Universal Robots URScript: Fase3.script

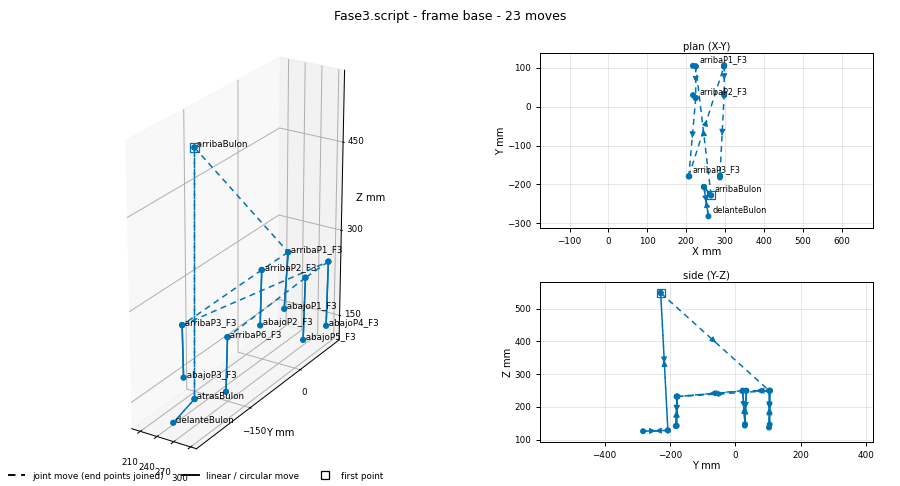
[picture p0: tool path of Fase3.script in frame base, 23 of 24 moves have a stored position in this frame; points joined in program order, loops and branches not executed]
def Fase3():
  set_tool_communication(True, 1000000, 2, 1, 1.5, 3.5)
  set_tool_output_mode(0)
  set_tool_digital_output_mode(0, 1)
  set_tool_digital_output_mode(1, 1)
  set_tool_voltage(0)
  set_safety_mode_transition_hardness(1)
  set_standard_analog_input_domain(0, 1)
  set_standard_analog_input_domain(1, 1)
  set_tool_analog_input_domain(0, 1)
  set_tool_analog_input_domain(1, 1)
  set_analog_outputdomain(0, 0)
  set_analog_outputdomain(1, 0)
  set_input_actions_to_default()
  set_tcp(p[0.00755148296704608,0.003639298738154023,0.026409592411711,0.0,0.0,0.0])
  set_payload(1.14, [0.022, -0.007, 0.054])
  set_gravity([0.0, 0.0, 9.82])
  step_count_833a9f29_8450_4b32_8ecf_da8deb8df3a1 = 0.0
  thread Step_Counter_Thread_0190bdf0_45ae_4d0e_b5b2_50c915833671():
    while (True):
      step_count_833a9f29_8450_4b32_8ecf_da8deb8df3a1 = step_count_833a9f29_8450_4b32_8ecf_da8deb8df3a1 + 1.0
      sync()
    end
  end
  run Step_Counter_Thread_0190bdf0_45ae_4d0e_b5b2_50c915833671()
  global Mesa=p[-0.3283222416297581,-0.20095078680444134,-0.01154506462095492,-2.1087277613487028,-2.3273776320839428,-7.166709239352482E-4]
  # begin: URCap Installation Node
  #   Source: Remote TCP & Toolpath, 1.2.65.build36, Universal Robots A/S
  #   Type: Remote TCP & Toolpath
  # end: URCap Installation Node
  # begin: URCap Installation Node
  #   Source: OnRobot, 5.1.6, OnRobot A/S
  #   Type: Configuración de OnRobot
  on_robot_type = 3
  on_robot_cycle = 2.0
  on_device_ip = "localhost"
  on_device_socket_port = 51234
  on_xmlrpc = rpc_factory("xmlrpc", "http://localhost:41414")
  on_RPC = rpc_factory("xmlrpc", "http://127.0.0.1:31416")
  ON_DEBUG_LOG = False
  on_isMetric = True
  on_toolConnector = True
  on_ioqc = False
  on_dual = False
  on_ft = False
  on_hex = False
  on_gecko = 0
  on_gripper = [False, False, False]
  #======    OnRobot Globals    ======#

  ON_MATH_PI=3.141593
  ON_ZEROPOSE=p[0.0,0.0,0.0,0.0,0.0,0.0]
  ON_ZEROFRAME=p[0.0,0.0,0.0,0.0,0.0,0.0]
  ON_ZERO3D=[0.0,0.0,0.0]
  ON_ZERO6D=[0.0,0.0,0.0,0.0,0.0,0.0]
  ON_ZERO8D=[0.0,0.0,0.0,0.0,0.0,0.0,0.0,0.0]
  ON_FALSE3D=[False,False,False]
  ON_FALSE6D=[False,False,False,False,False,False]
  ON_FALSE8D=[False,False,False,False,False,False,False,False]
  global on_return=0
  on_speedL=ON_ZERO6D
  on_speedBase=ON_ZERO6D
  on_speedVect=ON_ZERO6D
  on_speedExtra=ON_ZERO6D
  on_speedDC=ON_ZERO6D
  on_speedGecko=ON_ZERO6D
  on_floatRegShift=24
  on_intRegShift=24
  on_boolRegShift=64
  ON_BASE_SHIFT_FLOAT=24
  ON_BASE_SHIFT_INT=24
  ON_BASE_SHIFT_BOOL=64
  ON_DEVICE_SHIFT_FLOAT=3
  ON_DEVICE_SHIFT_INT=2
  ON_DEVICE_SHIFT_BOOL=7
  ON_COMMON_SHIFT_FLOAT=12
  ON_COMMON_SHIFT_INT=3
  ON_COMMON_SHIFT_BOOL=1
  ON_DI_SINGLE=0
  ON_DI_PRIMARY=1
  ON_DI_SECONDARY=2
  ON_DI_DUAL=3
  ON_DEVICE_ID_MISSING=0
  ON_INIT_TIMEOUT=500
  on_robot_TCP_offset=ON_ZEROFRAME
  on_tcp_offset_actual=ON_ZEROFRAME
  on_cog_actual=ON_ZEROFRAME
  on_mass_actual=0.0
  on_robot_mount=[0.0,0.0]

  #======    End of OnRobot Globals    ======#
  #======    OnRobot Interface Messages    ======#

  on_devices_primary_log="Dispositivos de OnRobot"
  on_devices_secondary_log="Dispositivo secundario de OnRobot"
  on_device_error_title="OnRobot - Error de dispositivo"
  on_install_error="La configuración de OnRobot no es correcta.<br>Compruebe el estado en la página de configuración de OnRobot, en la pestaña de instalación.<br>Programa detenido."
  on_device_missing="No hay ningún dispositivo conectado.<br>Programa detenido."
  ft_device_missing="No hay ningún sensor F/T OnRobot conectado.<br>Programa detenido."
  rg2ft_device_missing="No hay ninguna pinza RG2-FT conectada.<br>Programa detenido."
  rg_device_missing="No hay ninguna pinza RG conectada.<br>Programa detenido."
  vg_device_missing="No hay ninguna pinza VG conectada.<br>Programa detenido."
  gg_device_missing="No hay ninguna Gecko Gripper conectada.<br>Programa detenido."
  sg_device_missing="No hay ninguna Soft Gripper conectada.<br>Programa detenido."
  tfg_device_missing="No hay ninguna pinza 3FG conectada.<br>Programa detenido."
  on_xmlrpc_start_ip="Conexión al servidor XML-RPC de OnRobot:"
  on_java_comm_error_textmsg_title="OnRobot - Error de comunicación:"
  on_java_comm_controlsocket_open_error="Apertura de la toma 'javaSocket' incorrecta."
  on_java_comm_error_title="OnRobot - Error de comunicación"
  on_java_comm_socket_open_error="El establecimiento de la conexión con el URCap ha excedido el tiempo.<br>Compruebe el estado en la página de configuración de OnRobot, en la pestaña de instalación.<br>Programa detenido."
  on_rtde_feed_error_textmsg_title="OnRobot - Error de comunicación:"
  on_rtde_feed_open_error_textmsg="Apertura de la toma 'rtdeFeed' incorrecta."
  on_rtde_feed_error_title="OnRobot - Error de comunicación"
  on_rtde_feed_open_error="El establecimiento de la conexión con los dispositivos ha excedido el tiempo.<br>Asegúrese de que los dispositivos de OnRobot funcionen y compruebe el estado en la página de configuración de OnRobot, en la pestaña de instalación."

  #======    End of OnRobot Interface Messages    ======#
  #======    OnRobot Interface    ======#

  on_portopened_javaSocket=False
  on_rtde_feed_opened=False
  on_dataRead_running=False
  FT_SENSOR_ID_UNDEFINED=0
  FT_SENSOR_ID_UNKNOWN=1
  FT_SENSOR_ID_HEX_V1=11
  FT_SENSOR_ID_HEX_V2=12
  FT_SENSOR_ID_HEX_V3=13
  FT_SENSOR_ID_RG2FT_V0=20
  FT_SENSOR_ID_RG2FT_V1=21
  FT_SENSOR_ID_RG2FT_V2=22
  def on_error(status_flag,message,title,stop_var=False):
  if(status_flag):
  popup(message,title=title,error=True,blocking=False)
  stop_var=True
  end
  return stop_var
  end
  def on_warning(status_flag,message,title):
  if(status_flag):
  textmsg(title,message)
  end
  end
  def on_missing():
  popup(on_device_missing,title=on_device_error_title,error=True,blocking=False)
  halt
  end
  def ft_missing():
  popup(ft_device_missing,title=on_device_error_title,error=True,blocking=False)
  halt
  end
  def rg2ft_missing():
  popup(rg2ft_device_missing,title=on_device_error_title,error=True,blocking=False)
  halt
  end
  def rg_missing():
  popup(rg_device_missing,title=on_device_error_title,error=True,blocking=False)
  halt
  end
  def vg_missing():
  popup(vg_device_missing,title=on_device_error_title,error=True,blocking=False)
  halt
  end
  def gg_missing():
  popup(gg_device_missing,title=on_device_error_title,error=True,blocking=False)
  halt
  end
  def sg_missing():
  popup(sg_device_missing,title=on_device_error_title,error=True,blocking=False)
  halt
  end
  def tfg_missing():
  popup(tfg_device_missing,title=on_device_error_title,error=True,blocking=False)
  halt
  end
  def on_portclose_javaSocket():
  socket_close("javaSocket")
  on_portopened_javaSocket=False
  end
  def on_portopen_javaSocket():
  on_portclose_javaSocket()
  on_portopened_javaSocket=socket_open("127.0.0.1",44005,"javaSocket")
  if not on_portopened_javaSocket:
  textmsg(on_java_comm_error_textmsg_title,on_java_comm_controlsocket_open_error)
  popup(on_java_comm_socket_open_error,title=on_java_comm_error_title,error=True,blocking=False)
  halt
  end
  end
  def on_rtde_feed_close():
  socket_close("rtdeFeed")
  on_rtde_feed_opened=False
  end
  def on_rtde_feed_open():
  on_rtde_feed_close()
  on_rtde_feed_opened=socket_open(on_device_ip,on_device_socket_port,"rtdeFeed")
  if not on_rtde_feed_opened:
  on_rtde_feed_opened=socket_open(on_device_ip,on_device_socket_port,"rtdeFeed")
  end
  if not on_rtde_feed_opened:
  textmsg(on_rtde_feed_error_textmsg_title,on_rtde_feed_open_error_textmsg)
  popup(on_rtde_feed_open_error,title=on_rtde_feed_error_title,error=True,blocking=False)
  halt
  end
  end
  def on_dataRead():
  enter_critical
  floatRegDummy=read_input_float_register(0+on_floatRegShift)
  on_speedVect[0]=floatRegDummy/1000.0
  floatRegDummy=read_input_float_register(1+on_floatRegShift)
  on_speedVect[1]=floatRegDummy/1000.0
  floatRegDummy=read_input_float_register(2+on_floatRegShift)
  on_speedVect[2]=floatRegDummy/1000.0
  floatRegDummy=read_input_float_register(3+on_floatRegShift)
  on_speedVect[3]=floatRegDummy
  floatRegDummy=read_input_float_register(4+on_floatRegShift)
  on_speedVect[4]=floatRegDummy
  floatRegDummy=read_input_float_register(5+on_floatRegShift)
  on_speedVect[5]=floatRegDummy
  exit_critical
  end
  def on_set_rtde_watchdog(updateHz=5,ftWD=False,gripperWD=-1):
  local update_str=str_cat(" watchdog set to [Hz]: ",updateHz)
  if ftWD:
  watchdog_int_reg_str=str_cat("input_int_register_",0+on_intRegShift)
  rtde_set_watchdog(watchdog_int_reg_str,updateHz,"stop")
  if ON_DEBUG_LOG:
  textmsg(watchdog_int_reg_str,update_str)
  end
  end
  if not(gripperWD<0):
  if(gripperWD==ON_DI_SINGLE or gripperWD==ON_DI_PRIMARY or gripperWD==ON_DI_DUAL):
  watchdog_int_reg_str=str_cat("input_int_register_",3+on_intRegShift)
  rtde_set_watchdog(watchdog_int_reg_str,updateHz,"stop")
  if ON_DEBUG_LOG:
  textmsg(watchdog_int_reg_str,update_str)
  end
  end
  if(gripperWD==ON_DI_SECONDARY or gripperWD==ON_DI_DUAL):
  watchdog_int_reg_str=str_cat("input_int_register_",ON_DEVICE_SHIFT_INT+3+on_intRegShift)
  rtde_set_watchdog(watchdog_int_reg_str,updateHz,"stop")
  if ON_DEBUG_LOG:
  textmsg(watchdog_int_reg_str,update_str)
  end
  end
  end
  end
  def on_speedVect_get():
  return[on_speedVect[0],on_speedVect[1],on_speedVect[2],on_speedVect[3],on_speedVect[4],on_speedVect[5]]
  end
  def on_speedDC_get():
  local speedExtra=ON_ZERO6D
  if on_speedl_for_depthcompensation:
  speedExtra=[on_speedDC[0],on_speedDC[1],on_speedDC[2],on_speedDC[3],on_speedDC[4],on_speedDC[5]]
  end
  return speedExtra
  end
  def on_speedDC_set(speedDC):
  on_speedDC=[speedDC[0],speedDC[1],speedDC[2],speedDC[3],speedDC[4],speedDC[5]]
  end
  def on_speedGecko_get():
  local speedExtra=ON_ZERO6D
  if on_speedl_for_gecko:
  speedExtra=[on_speedGecko[0],on_speedGecko[1],on_speedGecko[2],on_speedGecko[3],on_speedGecko[4],on_speedGecko[5]]
  end
  return speedExtra
  end
  def on_speedGecko_set(speedGecko):
  on_speedGecko=[speedGecko[0],speedGecko[1],speedGecko[2],speedGecko[3],speedGecko[4],speedGecko[5]]
  end
  thread on_dataRead_thread():
  if ON_DEBUG_LOG:
  textmsg("Starting on_dataRead thread")
  end
  while on_dataRead_running:
  sync()
  on_dataRead()
  end
  if ON_DEBUG_LOG:
  textmsg("Stopping on_dataRead thread")
  end
  end

  #======    End of OnRobot Interface    ======#
  #======    OnRobot QC Setup Tool Connector    ======#

  def tc_setup_tool():
  if ON_DEBUG_LOG:
  textmsg("QC Setup Tool Connector start...")
  end
  set_tool_voltage(24)

  set_tool_communication(True,1000000,2,1,1.5,3.5)

  if ON_DEBUG_LOG:
  textmsg("QC Setup Tool Connector end.")
  end
  end

  #======    End of OnRobot QC Setup Tool Connector    ======#
  #======    OnRobot TCP Messages    ======#

  on_tcp_log_msg_default="OnRobot: Desplazamiento del TCP del robot establecido en:"
  on_tcp_log_msg_primary="OnRobot: Desplazamiento del TCP del robot establecido en primario:"
  on_tcp_log_msg_secondary="OnRobot: Desplazamiento del TCP del robot establecido en secundario:"

  #======    End of OnRobot TCP Messages    ======#
  #======    OnRobot TCP    ======#

  on_tcp_offset_actual=ON_ZEROFRAME
  on_tcp_offset_primary=ON_ZEROFRAME
  on_tcp_static_primary=ON_ZEROFRAME
  on_tcp_dynamic_primary=ON_ZEROFRAME
  on_tcp_vision_primary=ON_ZEROFRAME
  on_tcp_qc_primary=ON_ZEROFRAME
  on_tcp_base_primary=ON_ZEROFRAME
  on_tcp_gripper_static_primary=ON_ZEROFRAME
  on_tcp_tool_primary=ON_ZEROFRAME
  on_tcp_gripper_dynamic_primary=ON_ZEROFRAME
  on_tcp_gripper_primary=ON_ZEROFRAME
  on_tcp_offset_secondary=ON_ZEROFRAME
  on_tcp_static_secondary=ON_ZEROFRAME
  on_tcp_dynamic_secondary=ON_ZEROFRAME
  on_tcp_vision_secondary=ON_ZEROFRAME
  on_tcp_qc_secondary=ON_ZEROFRAME
  on_tcp_base_secondary=ON_ZEROFRAME
  on_tcp_gripper_static_secondary=ON_ZEROFRAME
  on_tcp_tool_secondary=ON_ZEROFRAME
  on_tcp_gripper_dynamic_secondary=ON_ZEROFRAME
  on_tcp_gripper_secondary=ON_ZEROFRAME
  def on_tcp_update_primary():
  if ON_DEBUG_LOG:
  textmsg("TCP Update Primary start..")
  end
  on_tcp_gripper_dynamic_primary=p[0.0, 0.0, 0.0, 0.0, 0.0, 0.0]
  enter_critical
  on_tcp_dynamic_primary=pose_trans(on_tcp_static_primary,on_tcp_gripper_dynamic_primary)
  on_tcp_offset_primary=pose_trans(on_tcp_dynamic_primary,on_tcp_tool_primary)
  exit_critical
  if ON_DEBUG_LOG:
  textmsg("TCP Update Primary end.")
  end
  end
  def on_tcp_init_primary():
  if ON_DEBUG_LOG:
  textmsg("TCP Init Primary start..")
  end
  enter_critical
  on_tcp_base_primary=pose_trans(on_tcp_vision_primary,on_tcp_qc_primary)
  on_tcp_static_primary=pose_trans(on_tcp_base_primary,on_tcp_gripper_static_primary)
  exit_critical
  on_tcp_update_primary()
  if ON_DEBUG_LOG:
  textmsg("TCP Init Primary end.")
  end
  end
  def on_tcp_offset_set(TCP_offset):
  if ON_DEBUG_LOG:
  textmsg("TCP Offset set started!")
  end
  on_tcp_offset_send(TCP_offset)
  if(on_follow_tcp):
  set_tcp(TCP_offset)
  end
  on_robot_TCP_offset=TCP_offset
  if ON_DEBUG_LOG:
  textmsg("TCP Offset set to: ",on_robot_TCP_offset)
  end
  end
  def on_tcp_offset_forced_set_actual(isPrimary=True):
  if(not on_follow_tcp):

  local tcp_log_msg=on_tcp_log_msg_default

  textmsg(tcp_log_msg,on_tcp_offset_actual)
  set_tcp(on_tcp_offset_actual)
  end
  end
  def on_tcp_update(isPrimary=True):
  on_tcp_update_primary()

  on_tcp_set_actual_to(isPrimary)
  end
  def on_tcp_set_actual_to(isPrimary=True):

  on_tcp_offset_actual=on_tcp_offset_primary
  if(on_follow_tcp):
  textmsg(on_tcp_log_msg_default,on_tcp_offset_actual)
  end

  on_tcp_active_is_primary=isPrimary
  on_tcp_offset_set(on_tcp_offset_actual)
  end
  def on_tcp_update_tool_primary(tool_offset):
  if ON_DEBUG_LOG:
  textmsg("TCP Update Tool Primary start..")
  end
  on_tcp_tool_primary=tool_offset
  on_tcp_update_primary()
  if ON_DEBUG_LOG:
  textmsg("TCP Update Tool Primary end.")
  end
  end
  def on_tcp_tool_rpy_get(xyz=[0.0,0.0,0.0],rpy=[0.0,0.0,0.0]):
  local rotvec=rpy2rotvec(rpy)
  local tool_offset=p[xyz[0],xyz[1],xyz[2],rotvec[0],rotvec[1],rotvec[2]]
  return tool_offset
  end

  def on_tcp_update_tool(tool_offset,tool_index=0):
  if ON_DEBUG_LOG:
  textmsg("TCP Update Tool start..")
  end
  if(tool_index!=ON_DI_SECONDARY):
  on_tcp_update_tool_primary(tool_offset)
  local isPrimary=True

  end
  on_tcp_set_actual_to(isPrimary)
  if ON_DEBUG_LOG:
  textmsg("TCP Update Tool end.")
  end
  end

  #======    End of OnRobot TCP    ======#
  #======    OnRobot Payload Messages    ======#

  on_mass_log_msg="OnRobot: Masa de la carga útil del robot establecida en:"
  on_cog_log_msg="OnRobot: Centro de gravedad de la carga útil del robot establecido en:"

  #======    End of OnRobot Payload Messages    ======#
  #======    OnRobot Payload    ======#

  on_cog_actual=ON_ZEROFRAME
  on_mass_actual=0.0
  on_cog_primary=ON_ZEROFRAME
  on_cog_L1L2_primary=ON_ZEROFRAME
  on_mass_primary=0.0
  on_mass_L1L2_primary=0.0
  on_cog_vision_primary=ON_ZEROFRAME
  on_cog_qc_primary=ON_ZEROFRAME
  on_cog_base_primary=ON_ZEROFRAME
  on_cog_gripper_primary=ON_ZEROFRAME
  on_cog_tool_primary=ON_ZEROFRAME
  on_mass_vision_primary=0.0
  on_mass_qc_primary=0.0
  on_mass_base_primary=0.0
  on_mass_gripper_primary=0.0
  on_mass_tool_primary=0.0
  on_cog_secondary=ON_ZEROFRAME
  on_mass_secondary=0.0
  on_cog_gripper_secondary=ON_ZEROFRAME
  on_mass_gripper_secondary=0.0
  on_cog_tool_secondary=ON_ZEROFRAME
  on_mass_tool_secondary=0.0
  ON_LB2KG001=0.45359237/100
  def on_payload_update_primary():
  if ON_DEBUG_LOG:
  textmsg("Payload Update Primary start..")
  end
  enter_critical
  on_mass_primary=on_mass_L1L2_primary+on_mass_tool_primary
  local massL1L2L3Ratio=on_mass_tool_primary/on_mass_primary
  local toolAbsCOG=pose_trans(on_tcp_dynamic_primary,on_cog_tool_primary)
  toolAbsCOG=p[toolAbsCOG[0],toolAbsCOG[1],toolAbsCOG[2],0.0,0.0,0.0]
  on_cog_primary=interpolate_pose(on_cog_L1L2_primary,toolAbsCOG,massL1L2L3Ratio)
  on_cog_primary=p[on_cog_primary[0],on_cog_primary[1],on_cog_primary[2],0.0,0.0,0.0]
  exit_critical
  if ON_DEBUG_LOG:
  textmsg("Payload Update Primary end.")
  end
  end
  def on_payload_init_primary():
  if ON_DEBUG_LOG:
  textmsg("Payload Init Primary start..")
  end
  enter_critical
  on_mass_base_primary=on_mass_vision_primary+on_mass_qc_primary
  local massL0L1Ratio=on_mass_qc_primary/on_mass_base_primary
  on_mass_L1L2_primary=on_mass_base_primary+on_mass_gripper_primary
  local massL1L2Ratio=on_mass_gripper_primary/on_mass_L1L2_primary
  local qcAbsCOG=pose_trans(on_tcp_vision_primary,on_cog_qc_primary)
  qcAbsCOG=p[qcAbsCOG[0],qcAbsCOG[1],qcAbsCOG[2],0.0,0.0,0.0]
  on_cog_base_primary=interpolate_pose(on_cog_vision_primary,qcAbsCOG,massL0L1Ratio)
  on_cog_base_primary=p[on_cog_base_primary[0],on_cog_base_primary[1],on_cog_base_primary[2],0.0,0.0,0.0]
  local gripperAbsCOG=pose_trans(on_tcp_base_primary,on_cog_gripper_primary)
  gripperAbsCOG=p[gripperAbsCOG[0],gripperAbsCOG[1],gripperAbsCOG[2],0.0,0.0,0.0]
  on_cog_L1L2_primary=interpolate_pose(on_cog_base_primary,gripperAbsCOG,massL1L2Ratio)
  on_cog_L1L2_primary=p[on_cog_L1L2_primary[0],on_cog_L1L2_primary[1],on_cog_L1L2_primary[2],0.0,0.0,0.0]
  exit_critical
  on_payload_update_primary()
  if ON_DEBUG_LOG:
  textmsg("Payload Init Primary end.")
  end
  end
  def on_payload_update():
  on_payload_update_primary()

  on_mass_actual =on_mass_primary
  on_cog_actual=on_cog_primary

  on_payload_set_actual()
  end
  def on_payload_set_actual():

  on_mass_actual =on_mass_primary
  on_cog_actual=on_cog_primary

  local CoG=[on_cog_actual[0],on_cog_actual[1],on_cog_actual[2]]
  on_payload_set(on_mass_actual,CoG)
  end
  def on_payload_update_tool_primary(tool_mass=0,tool_cog=[0.0,0.0,0.0]):
  if ON_DEBUG_LOG:
  textmsg("Payload Update Tool Primary start..")
  end
  on_cog_tool_primary=p[tool_cog[0],tool_cog[1],tool_cog[2],0.0,0.0,0.0]
  on_mass_tool_primary=tool_mass
  on_payload_update_primary()
  if ON_DEBUG_LOG:
  textmsg("Payload Update Tool Primary end.")
  end
  end
  def on_payload_set(mass,CoG):
  if ON_DEBUG_LOG:
  textmsg("Payload set started!")
  end
  local center_of_gravity=[CoG[0],CoG[1],CoG[2]]
  on_payload_send(center_of_gravity,mass)
  if(on_isMetric):
  local roundedMass=floor(mass*100+0.5)/100
  else:
  local roundedMass=floor(mass/ON_LB2KG001+0.5)*ON_LB2KG001
  end
  set_payload(roundedMass,center_of_gravity)
  on_mass_actual=roundedMass
  on_cog_actual=p[CoG[0],CoG[1],CoG[2],0.0,0.0,0.0]
  if ON_DEBUG_LOG:
  textmsg("Payload mass, CoG set to: ",str_cat(str_cat(mass,", "),CoG))
  end
  end

  def on_payload_update_secondary():
  end
  def on_payload_init_secondary():
  end

  def on_payload_update_tool(tool_mass,tool_cog=[0.0,0.0,0.0],tool_index=0):
  if ON_DEBUG_LOG:
  textmsg("Payload Update Tool start..")
  end
  if(tool_index!=ON_DI_SECONDARY):
  on_cog_tool_primary=p[tool_cog[0],tool_cog[1],tool_cog[2],0.0,0.0,0.0]
  on_mass_tool_primary=tool_mass
  else:
  on_cog_tool_secondary=p[tool_cog[0],tool_cog[1],tool_cog[2],0.0,0.0,0.0]
  on_mass_tool_secondary=tool_mass
  end
  on_payload_update()
  if ON_DEBUG_LOG:
  textmsg("Payload Update Tool end.")
  end
  end
  def on_payload_get_cog2tcp_tool(tool_index=0):
  if(tool_index!=ON_DI_SECONDARY):
  local cog_tool=[on_tcp_tool_primary[0],on_tcp_tool_primary[1],on_tcp_tool_primary[2]]
  else:
  local cog_tool=[on_tcp_tool_secondary[0],on_tcp_tool_secondary[1],on_tcp_tool_secondary[2]]
  end
  return cog_tool
  end

  #======    End of OnRobot Payload    ======#
  #======    OnRobot QC TCP    ======#

  onrobotmini=0

  def on_tcp_offset_send(TCP_offset):
  on_robot_TCP_offset=TCP_offset
  end
  def on_payload_send(CoG,mass):
  on_robot_payload_cog=CoG
  on_robot_payload_mass=mass
  end


  #======    End of OnRobot QC TCP    ======#
  #======    OnRobot  Speedl    ======#

  on_speedl_thread_handler=0
  on_speedl_is_enabled=False
  on_speedl_is_running=False
  on_speedl_acc=0.0
  ft_speedl_hg_caranteen_reached=False
  ft_speedl_hg_caranteen_safemode=False
  on_speedl_for_ftcontrol=False
  on_speedl_for_move=False
  on_speedl_for_handguide=False
  on_speedl_for_insertpart=False
  on_speedl_for_depthcompensation=False
  on_speedl_for_center=False
  on_speedl_for_gecko=False
  on_speedl_acc=10000.0
  on_speedl_acc_to_zero=3.0
  ON_SPEEDL_FTCONTROL=1
  ON_SPEEDL_HANDGUIDE=2
  ON_SPEEDL_MOVE=3
  ON_SPEEDL_INSERTPART=4
  ON_SPEEDL_DEPTHCOMP=5
  ON_SPEEDL_CENTER=6
  ON_SPEEDL_GECKO=7
  def on_speedl_add_extra(speedBase,speedExtra):
  speedSum=ON_ZERO6D
  speedBaseP=p[speedBase[0],speedBase[1],speedBase[2],speedBase[3],speedBase[4],speedBase[5]]
  speedExtraP=p[speedExtra[0],speedExtra[1],speedExtra[2],speedExtra[3],speedExtra[4],speedExtra[5]]
  speedSumP=pose_add(speedExtraP,speedBaseP)
  speedSum=[speedSumP[0],speedSumP[1],speedSumP[2],speedSumP[3],speedSumP[4],speedSumP[5]]
  return speedSum
  end

  thread on_speedl_thread():
  if ON_DEBUG_LOG:
  textmsg("Speedl thread started..")
  end
  enter_critical
  on_speedl_is_running=True
  on_speedl_is_enabled=True
  exit_critical
  on_speedL=ON_ZERO6D

  while on_speedl_is_running:
  on_speedBase=on_speedVect_get()
  on_speedL=on_speedBase



  if on_speedl_is_enabled:
  speedl(on_speedL,a=on_speedl_acc,t=0.001)
  else:
  speedl(ON_ZERO6D,a=on_speedl_acc_to_zero,t=0.001)
  end
  end

  on_speedL=ON_ZERO6D
  if ON_DEBUG_LOG:
  textmsg("Speedl thread ended.")
  end
  end
  def on_speedl_integer_get():
  local speedl_integer=binary_list_to_integer([on_speedl_for_ftcontrol,on_speedl_for_handguide,on_speedl_for_move,on_speedl_for_insertpart,on_speedl_for_depthcompensation,on_speedl_for_center,on_speedl_for_gecko])
  return speedl_integer
  end
  def on_speedl_start_for(speedl_id):
  if(speedl_id==ON_SPEEDL_FTCONTROL):
  on_speedl_for_ftcontrol=True
  elif(speedl_id==ON_SPEEDL_HANDGUIDE):
  on_speedl_for_handguide=True
  elif(speedl_id==ON_SPEEDL_MOVE):
  on_speedl_for_move=True
  elif(speedl_id==ON_SPEEDL_INSERTPART):
  on_speedl_for_insertpart=True
  elif(speedl_id==ON_SPEEDL_DEPTHCOMP):
  on_speedl_for_depthcompensation=True
  elif(speedl_id==ON_SPEEDL_CENTER):
  on_speedl_for_center=True
  elif(speedl_id==ON_SPEEDL_GECKO):
  on_speedl_for_gecko=True
  else:
  textmsg("Unknown Start speedl ID received: ",speedl_id)
  end
  local speedl_integer=on_speedl_integer_get()
  if not(speedl_integer==0):
  if not on_speedl_is_running:
  on_speedl_thread_handler=run on_speedl_thread()
  end
  end
  return on_speedl_is_running
  end
  def on_speedl_stop_for(speedl_id,brake=10):
  if(speedl_id==ON_SPEEDL_FTCONTROL):
  on_speedl_for_ftcontrol=False
  elif(speedl_id==ON_SPEEDL_HANDGUIDE):
  on_speedl_for_handguide=False
  elif(speedl_id==ON_SPEEDL_MOVE):
  on_speedl_for_move=False
  elif(speedl_id==ON_SPEEDL_INSERTPART):
  on_speedl_for_insertpart=False
  elif(speedl_id==ON_SPEEDL_DEPTHCOMP):
  on_speedl_for_depthcompensation=False
  on_speedDC_set(ON_ZERO6D)
  elif(speedl_id==ON_SPEEDL_CENTER):
  on_speedl_for_center=False
  elif(speedl_id==ON_SPEEDL_GECKO):
  on_speedl_for_gecko=False
  on_speedGecko_set(ON_ZERO6D)
  else:
  textmsg("Unknown Stop speedl ID received: ",speedl_id)
  end
  local speedl_integer=on_speedl_integer_get()
  if(speedl_integer==0):
  if(on_speedl_is_running):
  kill on_speedl_thread_handler
  enter_critical
  on_speedl_is_running=False
  exit_critical

  end
  if ON_DEBUG_LOG:
  textmsg("Speedl thread stopped")
  end
  stopl(brake)
  end
  return on_speedl_is_running
  end
  def on_speedl_pause():
  on_speedl_is_enabled=False
  return on_speedl_integer_get()
  end
  def on_speedl_resume():
  on_speedl_is_enabled=True
  return on_speedl_integer_get()
  end
  def on_wait_ms(time_ms):
  local sync_time=ceil(norm(time_ms/2.0))
  while(sync_time>0):
  sync_time=sync_time-1
  sync()
  end
  end

  #======    End of OnRobot  Speedl    ======#
  on_install_tcp = False
  on_follow_tcp = False
  textmsg(on_devices_primary_log, ": Quick Changer + Lado de la herramienta de QC + [0.0, 0.0, 0.0, 0.0, 0.0, 0.0]")
  on_tcp_active_is_primary = True
  on_tcp_vision_primary = p[0.0, 0.0, 0.0, 0.0, 0.0, 0.0]
  on_cog_vision_primary = p[0.0, 0.0, 0.0, 0.0, 0.0, 0.0]
  on_mass_vision_primary = 0.0
  on_tcp_qc_primary = p[0.0, 0.0, 0.0136, 0.0, 0.0, 0.0]
  on_cog_qc_primary = p[0.0, 0.0, 0.004, 0.0, 0.0, 0.0]
  on_mass_qc_primary = 0.06
  on_tcp_gripper_static_primary = p[0.0, 0.0, 0.017, 0.0, 0.0, 0.0]
  on_cog_gripper_primary = p[0.0, 0.0, 0.002, 0.0, 0.0, 0.0]
  on_mass_gripper_primary = 0.14
  on_tcp_tool_primary = p[0.0, 0.0, 0.0, 0.0, 0.0, 0.0]
  on_cog_tool_primary = p[0.0, 0.0, 0.0, 0.0, 0.0, 0.0]
  on_mass_tool_primary = 0.0
  #======    OnRobot Run    ======#

  textmsg(on_xmlrpc_start_ip,on_device_ip)
  on_portopen_javaSocket()
  sync()
  on_rtde_feed_open()
  sync()
  local gripperWDs=binary_list_to_integer(on_gripper)
  if gripperWDs==0:
  gripperWDs=-1
  else:
  gripperWDs=floor(gripperWDs/2)
  end
  on_set_rtde_watchdog(updateHz=0.2,ftWD=on_ft,gripperWD=gripperWDs)
  sync()
  on_dataRead_running=True
  sync()
  on_dataRead_thrd=run on_dataRead_thread()
  sync()
  on_tcp_init_primary()
  on_payload_init_primary()

  on_tcp_set_actual_to(on_tcp_active_is_primary)
  if(on_follow_tcp):
  on_payload_set_actual()
  end

  #======    End of OnRobot Run    ======#
  #======    OnRobot QC Start    ======#

  if(on_toolConnector):
  tc_setup_tool()
  end
  sync()

  #======    End of OnRobot QC Start    ======#
  # end: URCap Installation Node
  global arribaBulon_p=p[.264097371719, -.228254341384, .548494258749, 1.585288091520, .085368942758, .052684265010]
  global arribaBulon_q=[0.0823671817779541, -1.5479493898204382, -0.842977762222274, -2.249339719811945, 0.01133561134338383, -1.6629841963397176]
  global atrasBulon_p=p[.245619565393, -.206229029031, .127949595254, 1.145266979799, 1.284974715224, -1.172261599952]
  global atrasBulon_q=[0.18570303241219666, -1.8425440913304127, -2.1757274455361326, -2.137330201992251, 0.1096066770252433, -1.7350318094075643]
  global delanteBulon_p=p[.257367062930, -.282169444566, .125542628574, 1.158631853822, 1.223105278388, -1.250786556870]
  global delanteBulon_q=[-0.127409035395587, -2.02615272864022, -1.95040543910366, -2.0546015954477355, -0.14137166941154078, -1.8664551020827291]
  global arribaP1_F3_p=p[.224644079235, .103836313498, .249354312056, -2.208051583079, -2.214597805453, .012045887033]
  global arribaP1_F3_q=[0.9707521299592239, -1.174781119517391, -2.0064305080926808, -1.5350170771289937, 1.5830136315588959, -2.1699678590045597]
  global abajoP1_F3_p=p[.217351130895, .105158373635, .145871126277, -2.208007269394, -2.214589077087, .011773755537]
  global abajoP1_F3_q=[1.0053096491487898, -1.3109168011728976, -2.4436354857172944, -0.9609782861480696, 1.5838862961847608, -2.1366320702914097]
  global arribaP2_F3_p=p[.224582479854, .022513190074, .249352391909, -2.207989835995, -2.214569210422, .012088793108]
  global arribaP2_F3_q=[0.6852162643329649, -1.0683160351457337, -2.0586158527273106, -1.5934856070708179, 1.5814428352320764, -2.455329191705632]
  global abajoP2_F3_p=p[.217746809497, .029725857966, .147153686199, -2.207987963195, -2.214642841298, .012082484581]
  global abajoP2_F3_q=[0.7419977188110352, -1.1732912820628645, -2.511789321899414, -1.0345638555339338, 1.5826172828674319, -2.399748627339495]
  global arribaP3_F3_p=p[.206750338136, -.179228225553, .231443959029, -2.197588078884, 2.235277736991, -.020786326198]
  global arribaP3_F3_q=[-0.18465583486099035, -1.3281955607676812, -2.0006709215611025, -1.3676400018627604, 1.5652112731884946, -0.1644100155378494]
  global abajoP3_F3_p=p[.208204529507, -.179202485408, .142240823155, -2.197553268895, 2.235243844556, -.020796942752]
  global abajoP3_F3_q=[-0.18301994005315336, -1.5208934110454173, -2.310643196105966, -0.8649354738047563, 1.565710783004826, -0.16392451921577944]
  global arribaP4_F3_p=p[.297933427712, .105957309290, .249359521855, -2.208163486704, -2.214602719616, .012089079617]
  global arribaP4_F3_q=[0.7490953149560091, -1.5138985931798459, -1.7521360360771503, -1.4535102010608423, 1.5802211047555632, -2.392322805708589]
  global abajoP4_F3_p=p[.297416304891, .103134700907, .136772641869, -2.207987172695, -2.214699703310, .011928594507]
  global abajoP4_F3_q=[0.7431611954992511, -1.7071065413756177, -2.13331594471272, -0.8791223442295077, 1.5809192364563067, -2.3998277214921577]
  global arribaP5_F3_p=p[.297927188132, .033813878502, .249377734153, -2.208173548754, -2.214589723707, .011925302641]
  global arribaP5_F3_q=[0.5391322059410543, -1.4463543511276873, -1.8116517635701346, -1.4641567094980132, 1.5784757755036594, -2.6021113817983164]
  global abajoP5_F3_p=p[.297930409515, .029154935950, .142651108607, -2.208220572640, -2.214607723347, .011878116817]
  global abajoP5_F3_q=[0.524354457855229, -1.6304494343199663, -2.1841697692871014, -0.907690839176535, 1.5789034366607568, -2.6182459036456485]
  global arribaP6_F3_p=p[.286922377788, -.177452737853, .231463994865, -2.197503334999, 2.235293632857, -.020976529593]
  global arribaP6_F3_q=[-0.13142329267507336, -1.6315337847643132, -1.7285740911751137, -1.3363986082522743, 1.5632914110110594, -0.11187560505271055]
  global abajoP6_F3_p=p[.286936793143, -.182063295540, .141255559416, -2.197478510061, 2.235221511214, -.020803429330]
  global abajoP6_F3_q=[-0.1460840583919243, -1.8058921770385403, -1.9922933411515018, -0.8983209660015365, 1.564164075637315, -0.12775810124598674]
  $ 1 "Robot Program"
  $ 2 "Set DO[0]=Apagar"
  set_standard_digital_out(0, False)
  $ 3 "i≔1"
  global i=1
  $ 4 "Loop i≤6"
  while (i <= 6):
    $ 5 "MoveJ"
    $ 6 "arribaBulon" "breakAfter"
    movej(get_inverse_kin(arribaBulon_p, qnear=arribaBulon_q), a=1.2, v=0.75)
    $ 7 "MoveJ"
    $ 8 "atrasBulon" "breakAfter"
    movej(get_inverse_kin(atrasBulon_p, qnear=atrasBulon_q), a=1.2, v=0.75)
    $ 9 "MoveJ"
    $ 10 "delanteBulon" "breakAfter"
    movej(get_inverse_kin(delanteBulon_p, qnear=delanteBulon_q), a=1.3962634015954636, v=1.0471975511965976)
    $ 11 "Set DO[0]=Encender"
    set_standard_digital_out(0, True)
    $ 12 "Wait: 0.25"
    sleep(0.25)
    $ 13 "MoveJ"
    $ 14 "atrasBulon" "breakAfter"
    movej(get_inverse_kin(atrasBulon_p, qnear=atrasBulon_q), a=1.3962634015954636, v=1.0471975511965976)
    $ 15 "MoveJ"
    $ 16 "arribaBulon" "breakAfter"
    movej(get_inverse_kin(arribaBulon_p, qnear=arribaBulon_q), a=1.2, v=0.75)
    $ 17 "If i≟1"
    if (i == 1):
      $ 18 "MoveJ"
      $ 19 "arribaP1_F3" "breakAfter"
      movej(get_inverse_kin(arribaP1_F3_p, qnear=arribaP1_F3_q), a=1.2, v=0.75)
      $ 20 "MoveL"
      $ 21 "abajoP1_F3" "breakAfter"
      movel(abajoP1_F3_p, a=1.2, v=0.25)
      $ 22 "Wait: 0.25"
      sleep(0.25)
      $ 23 "Set DO[0]=Apagar"
      set_standard_digital_out(0, False)
      $ 24 "MoveL"
      $ 25 "arribaP1_F3" "breakAfter"
      movel(arribaP1_F3_p, a=1.2, v=0.25)
    else:
      $ 26 "ElseIf i≟2"
      if (i == 2):
        $ 27 "MoveJ"
        $ 28 "arribaP2_F3" "breakAfter"
        movej(get_inverse_kin(arribaP2_F3_p, qnear=arribaP2_F3_q), a=1.3962634015954636, v=1.0471975511965976)
        $ 29 "MoveL"
        $ 30 "abajoP2_F3" "breakAfter"
        movel(abajoP2_F3_p, a=1.2, v=0.25)
        $ 31 "Wait: 0.25"
        sleep(0.25)
        $ 32 "Set DO[0]=Apagar"
        set_standard_digital_out(0, False)
        $ 33 "MoveL"
        $ 34 "arribaP2_F3" "breakAfter"
        movel(arribaP2_F3_p, a=1.2, v=0.25)
      else:
        $ 35 "ElseIf i≟3"
        if (i == 3):
          $ 36 "MoveJ"
          $ 37 "arribaP3_F3" "breakAfter"
          movej(get_inverse_kin(arribaP3_F3_p, qnear=arribaP3_F3_q), a=1.3962634015954636, v=1.0471975511965976)
          $ 38 "MoveL"
          $ 39 "abajoP3_F3" "breakAfter"
          movel(abajoP3_F3_p, a=1.2, v=0.25)
          $ 40 "Wait: 0.25"
          sleep(0.25)
          $ 41 "Set DO[0]=Apagar"
          set_standard_digital_out(0, False)
          $ 42 "MoveL"
          $ 43 "arribaP3_F3" "breakAfter"
          movel(arribaP3_F3_p, a=1.2, v=0.25)
        else:
          $ 44 "ElseIf i≟4"
          if (i == 4):
            $ 45 "MoveJ"
            $ 46 "arribaP4_F3" "breakAfter"
            movej(get_inverse_kin(arribaP4_F3_p, qnear=arribaP4_F3_q), a=1.3962634015954636, v=1.0471975511965976)
            $ 47 "MoveL"
            $ 48 "abajoP4_F3" "breakAfter"
            movel(abajoP4_F3_p, a=1.2, v=0.25)
            $ 49 "Wait: 0.25"
            sleep(0.25)
            $ 50 "Set DO[0]=Apagar"
            set_standard_digital_out(0, False)
            $ 51 "MoveL"
            $ 52 "arribaP4_F3" "breakAfter"
            movel(arribaP4_F3_p, a=1.2, v=0.25)
          else:
            $ 53 "ElseIf i≟5"
            if (i == 5):
              $ 54 "MoveJ"
              $ 55 "arribaP5_F3" "breakAfter"
              movej(get_inverse_kin(arribaP5_F3_p, qnear=arribaP5_F3_q), a=1.3962634015954636, v=1.0471975511965976)
              $ 56 "MoveL"
              $ 57 "abajoP5_F3" "breakAfter"
              movel(abajoP5_F3_p, a=1.2, v=0.25)
              $ 58 "Wait: 0.25"
              sleep(0.25)
              $ 59 "Set DO[0]=Apagar"
              set_standard_digital_out(0, False)
              $ 60 "MoveL"
              $ 61 "arribaP5_F3" "breakAfter"
              movel(arribaP5_F3_p, a=1.2, v=0.25)
            else:
              $ 62 "ElseIf i≟6"
              if (i == 6):
                $ 63 "MoveJ"
                $ 64 "arribaP6_F3" "breakAfter"
                movej(get_inverse_kin(arribaP6_F3_p, qnear=arribaP6_F3_q), a=1.3962634015954636, v=1.0471975511965976)
                $ 65 "MoveL"
                $ 66 "abajoP6_F3" "breakAfter"
                movel(abajoP6_F3_p, a=1.2, v=0.25)
                $ 67 "Wait: 0.25"
                sleep(0.25)
                $ 68 "Set DO[0]=Apagar"
                set_standard_digital_out(0, False)
                $ 69 "MoveL"
                $ 70 "arribaP6_F3" "breakAfter"
                movel(arribaP6_F3_p, a=1.2, v=0.25)
              end
            end
          end
        end
      end
    end
    $ 71 "NumPiezas≔i"
    global NumPiezas=i
    $ 72 "i≔i+1"
    global i=i+1
  end
  $ 73 "Home"
  movej([0.0, -1.5707963267948966, 0.0, -1.5707963267948966, 0.0, 0.0], a=1.3962634015954636, v=1.0471975511965976)
end
